(* Logix 5000 project; controller Savage_Saw vendor 1 type 14 code 152 rev 37.11; software revision 37.01 *)

TASK MainTask (continuous, watchdog 500 ms) : MainProgram, Inputs

MODULES
   Local : vendor 1 type 14 code 152 (PointIO 0, rev 37.11)
      Kane : vendor 590 type 43 code 5 (Ethernet 192.168.3.12, rev 1.1, StandardDataDriven RPI 20 ms, StandardDataDriven RPI 20 ms)
      RemoteHPU : 1734-AENTR (Ethernet 192.168.3.11, rev 7.13, Output RPI 20 ms)
         AnalogIn5_6 : 1734-IE2V (PointIO 1, rev 3.5, Input RPI 80 ms)
         InputDC0_8 : 1734-IB8 (PointIO 2, rev 3.22)
         InputDC9_15 : 1734-IB8 (PointIO 3, rev 3.1)
         OutputDC0_3 : vendor 1 type 7 code 134 (PointIO 5, rev 3.2)
         OutputDC4_7 : vendor 1 type 7 code 134 (PointIO 6, rev 3.2)
      Analog0_1 : 1734-IE2V (PointIO 2, rev 3.5, Input RPI 80 ms)
      Analog2_3 : 1734-IE2V (PointIO 3, rev 3.4, Input RPI 80 ms)
      Analog4_5 : 1734-IE2V (PointIO 4, rev 3.1, Input RPI 80 ms)
      Discrete_IO : Embedded (PointIO 1, rev 37.11, Output RPI 20 ms)
      SpindleControl : 1734-OE2V (PointIO 5, rev 3.1, Output RPI 80 ms)
       : 1734-OA4 (PointIO 6, rev 3.22, Output RPI 20 ms)
       : 1734-OA4 (PointIO 7, rev 3.1, Output RPI 20 ms)
       : 1734-OA4 (PointIO 8, rev 3.1, Output RPI 20 ms)
END_MODULES

TYPE AxisData :
STRUCT
   PositionActual : REAL;
   PositionCommand : REAL;
   VelocityCommand : REAL;
   InPosition : BOOL;
   AtVelocity : BOOL;
   OpenLoop : BOOL;
   FaultInput : BOOL;
   LimitPos : BOOL;
   LimitNeg : BOOL;
   Stopped : BOOL;
   InputEstimated : BOOL;
   OutputEnabled : BOOL;
   TargetGeneratorDone : BOOL;
   TargetGeneratorStateA : BOOL;
   TargetGeneratorStateB : BOOL;
   DirectOutput : BOOL;
   Enabled : BOOL;
   ExternalHalt : BOOL;
   Halted : BOOL;
   ForceControlled : BOOL;
   ForceLimitEnabled : BOOL;
   ForceLimited : BOOL;
   AtForce : BOOL;
   ForceInputEstimated : BOOL;
   ForceTargetGeneratorDone : BOOL;
   ForceTargetGeneratorStateA : BOOL;
   ForceTargetGeneratorStateB : BOOL;
   TargetGeneratorBusy : BOOL;
   ForceTargetGeneratorBusy : BOOL;
   FeedbackOK : BOOL;
   FeedbackOkSecondary : BOOL;
   StateMachineEnabled : BOOL;
   zs29 : BOOL;
   zs30 : BOOL;
   CommandAcknowledged : BOOL;
   CommandMove : BOOL;
   CommandJog : BOOL;
   Reverse : BOOL;
   z03 : BOOL;
   z04 : BOOL;
   z05 : BOOL;
   z06 : BOOL;
   z07 : BOOL;
   z08 : BOOL;
   z09 : BOOL;
   z10 : BOOL;
   z11 : BOOL;
   z12 : BOOL;
   z13 : BOOL;
   z14 : BOOL;
   z15 : BOOL;
   z16 : BOOL;
   z17 : BOOL;
   z18 : BOOL;
   z19 : BOOL;
   z20 : BOOL;
   z21 : BOOL;
   z22 : BOOL;
   z23 : BOOL;
   z24 : BOOL;
   z25 : BOOL;
   z26 : BOOL;
   z27 : BOOL;
   z28 : BOOL;
   z29 : BOOL;
   z30 : BOOL;
   z31 : BOOL;
END_STRUCT
END_TYPE

VAR_GLOBAL   (* controller tags *)
   Axis : AxisData[3];
   InBackGaugePot : ALIAS FOR Local:3:I.Ch1Data;
   inMS1HydraulicPump : ALIAS FOR Local:1:I.Data.1;
   inMS2HydraulicLoopPump : ALIAS FOR Local:1:I.Data.2;
   InMS3HydCoolingFan : ALIAS FOR Local:1:I.Data.3;
   inMS4CoolantPump : ALIAS FOR Local:1:I.Data.4;
   inMS5SwarfPump : ALIAS FOR Local:1:I.Data.5;
   inMS6SwarfConveyor : ALIAS FOR Local:1:I.Data.6;
   inRaiseLowerPot : ALIAS FOR Local:2:I.Ch1Data;
   inSpindleAside : ALIAS FOR Local:4:I.Ch0Data;
   inSpindleBside : ALIAS FOR Local:4:I.Ch1Data;
   inSpindleSpeed : ALIAS FOR Local:2:I.Ch0Data;
   inSR1SafetyRelay : ALIAS FOR Local:1:I.Data.0;
   inTraversePot : ALIAS FOR Local:3:I.Ch0Data;
   outLaserLine : ALIAS FOR Local:8:O.Data.0;
   outMS1HydraulicPump : ALIAS FOR Local:6:O.Data.0;
   outMS2HydraulicLoopPump : ALIAS FOR Local:6:O.Data.1;
   outMS3HydraulicCoolingFan : ALIAS FOR Local:6:O.Data.2;
   outMS4CoolantPump : ALIAS FOR Local:6:O.Data.3;
   outMS5SwarfPump : ALIAS FOR Local:7:O.Data.0;
   outMS6SwarfConveyor : ALIAS FOR Local:7:O.Data.1;
   outSpindleMotor : ALIAS FOR Local:5:O.Ch1Data;
   outSpindlePump : ALIAS FOR Local:5:O.Ch0Data;
   outStackLtAmber : ALIAS FOR Local:8:O.Data.2;
   outStackLtGreen : ALIAS FOR Local:8:O.Data.1;
   outStackLtRed : ALIAS FOR Local:8:O.Data.3;
   tbA1JogIn : BOOL;
   tbA1JogOut : BOOL;
   tbA2JogMinus : BOOL;
   tbA3JogMinus : BOOL;
   tbA3JogPlus : BOOL;
   tbAutoCut : BOOL;
   tbAutoGage : BOOL;
   tbAutoWet : BOOL;
   tbBladeChange : BOOL;
   tbBladeCompensation : BOOL;
   tbBladeMeasure : BOOL;
   tbCCW : BOOL;
   tbCoolant : BOOL;
   tbCW : BOOL;
   tbDryBump : BOOL;
   tbDryDist : BOOL;
   tbLaser : BOOL;
   tbMS1HydPump : BOOL;
   tbMS2LoopPump : BOOL;
   tbMS3HydCoolingFan : BOOL;
   tbMS4CoolantPump : BOOL;
   tbMS5SwarfPump : BOOL;
   tbMS6SwarfConveyor : BOOL;
   tbNorthRef : BOOL;
   tbOnOff : BOOL;
   tbPlateMeasure : BOOL;
   tbSouthRef : BOOL;
   tbWetBump : BOOL;
   tbWetDistance : BOOL;
   test : DINT;
   tmrTest : TIMER := (PRE := 1000);
   X_AutoCut : BOOL;
   X_AutoGauge : BOOL;
   X_BladeChange : BOOL;
   X_BladeMeasure : BOOL;
   X_Fault : BOOL;
   X_Homing : BOOL;
   X_Manual : BOOL;
   X_Off : BOOL;
END_VAR

PROGRAM Inputs   (* main routine Main *)

ROUTINE inAnalog   (* ladder *)
   0: ;
END_ROUTINE

ROUTINE Main   (* ladder *)
END_ROUTINE
END_PROGRAM

PROGRAM MainProgram   (* main routine Main *)
VAR
   iAxis : DINT;
END_VAR

ROUTINE Main   (* ladder *)
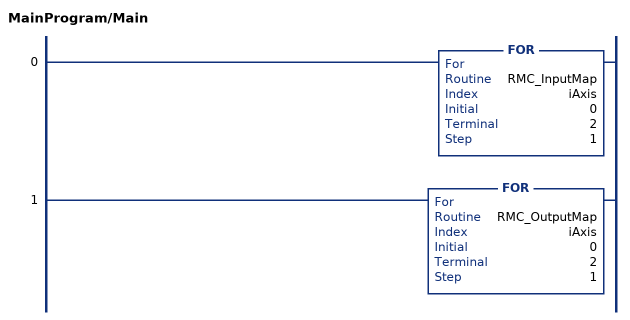
   0: FOR(RMC_InputMap,iAxis,0,2,1);
   1: FOR(RMC_OutputMap,iAxis,0,2,1);
END_ROUTINE

ROUTINE RMC_InputMap   (* ladder *)
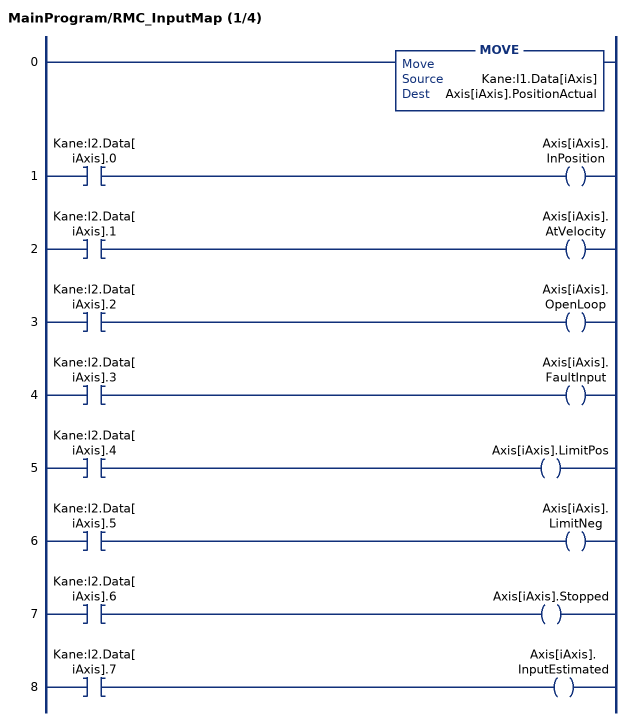
   0: MOVE(Kane:I1.Data[iAxis],Axis[iAxis].PositionActual);
   1: XIC(Kane:I2.Data[iAxis].0)OTE(Axis[iAxis].InPosition);
   2: XIC(Kane:I2.Data[iAxis].1)OTE(Axis[iAxis].AtVelocity);
   3: XIC(Kane:I2.Data[iAxis].2)OTE(Axis[iAxis].OpenLoop);
   4: XIC(Kane:I2.Data[iAxis].3)OTE(Axis[iAxis].FaultInput);
   5: XIC(Kane:I2.Data[iAxis].4)OTE(Axis[iAxis].LimitPos);
   6: XIC(Kane:I2.Data[iAxis].5)OTE(Axis[iAxis].LimitNeg);
   7: XIC(Kane:I2.Data[iAxis].6)OTE(Axis[iAxis].Stopped);
   8: XIC(Kane:I2.Data[iAxis].7)OTE(Axis[iAxis].InputEstimated);
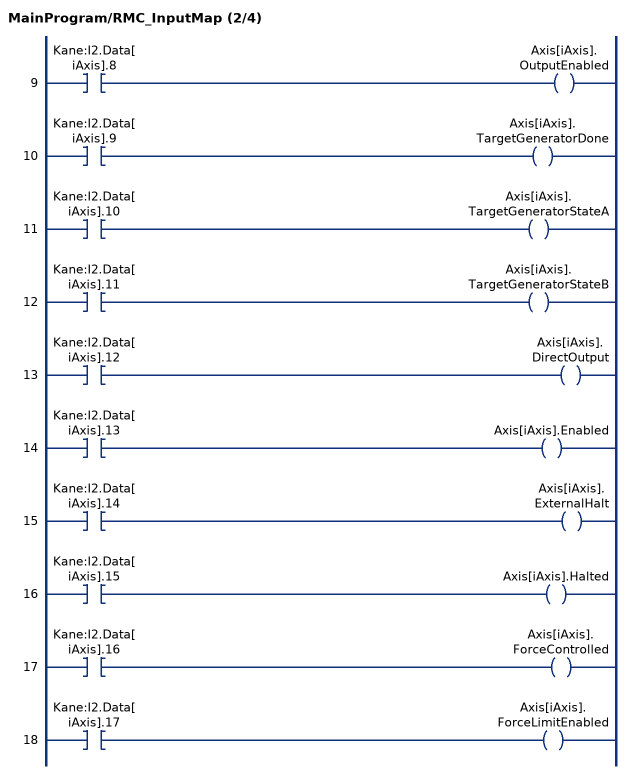
   9: XIC(Kane:I2.Data[iAxis].8)OTE(Axis[iAxis].OutputEnabled);
   10: XIC(Kane:I2.Data[iAxis].9)OTE(Axis[iAxis].TargetGeneratorDone);
   11: XIC(Kane:I2.Data[iAxis].10)OTE(Axis[iAxis].TargetGeneratorStateA);
   12: XIC(Kane:I2.Data[iAxis].11)OTE(Axis[iAxis].TargetGeneratorStateB);
   13: XIC(Kane:I2.Data[iAxis].12)OTE(Axis[iAxis].DirectOutput);
   14: XIC(Kane:I2.Data[iAxis].13)OTE(Axis[iAxis].Enabled);
   15: XIC(Kane:I2.Data[iAxis].14)OTE(Axis[iAxis].ExternalHalt);
   16: XIC(Kane:I2.Data[iAxis].15)OTE(Axis[iAxis].Halted);
   17: XIC(Kane:I2.Data[iAxis].16)OTE(Axis[iAxis].ForceControlled);
   18: XIC(Kane:I2.Data[iAxis].17)OTE(Axis[iAxis].ForceLimitEnabled);
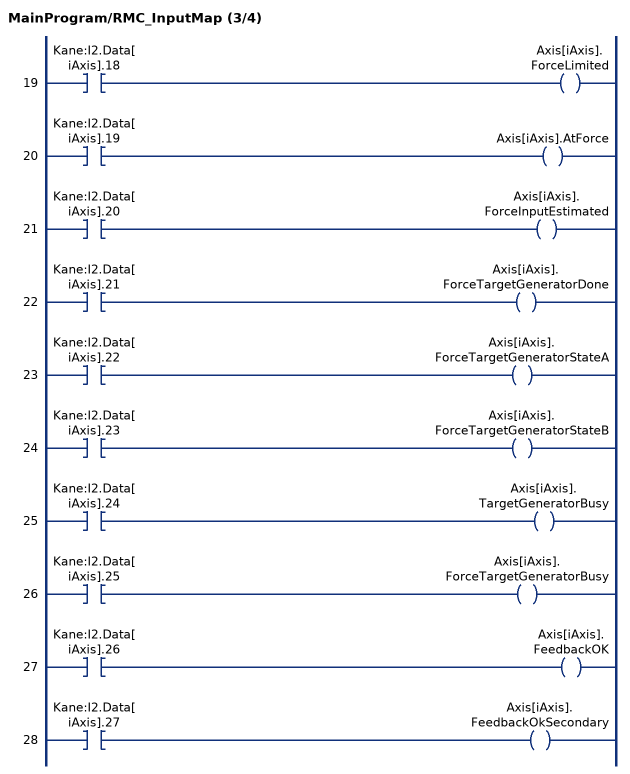
   19: XIC(Kane:I2.Data[iAxis].18)OTE(Axis[iAxis].ForceLimited);
   20: XIC(Kane:I2.Data[iAxis].19)OTE(Axis[iAxis].AtForce);
   21: XIC(Kane:I2.Data[iAxis].20)OTE(Axis[iAxis].ForceInputEstimated);
   22: XIC(Kane:I2.Data[iAxis].21)OTE(Axis[iAxis].ForceTargetGeneratorDone);
   23: XIC(Kane:I2.Data[iAxis].22)OTE(Axis[iAxis].ForceTargetGeneratorStateA);
   24: XIC(Kane:I2.Data[iAxis].23)OTE(Axis[iAxis].ForceTargetGeneratorStateB);
   25: XIC(Kane:I2.Data[iAxis].24)OTE(Axis[iAxis].TargetGeneratorBusy);
   26: XIC(Kane:I2.Data[iAxis].25)OTE(Axis[iAxis].ForceTargetGeneratorBusy);
   27: XIC(Kane:I2.Data[iAxis].26)OTE(Axis[iAxis].FeedbackOK);
   28: XIC(Kane:I2.Data[iAxis].27)OTE(Axis[iAxis].FeedbackOkSecondary);
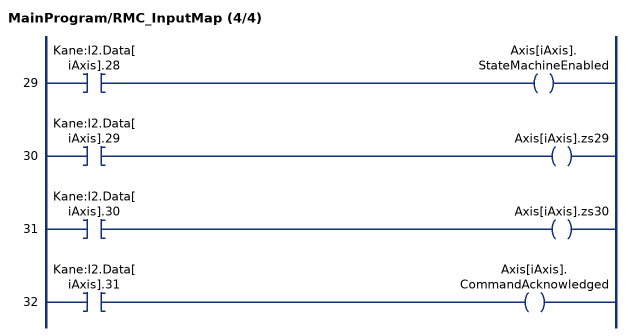
   29: XIC(Kane:I2.Data[iAxis].28)OTE(Axis[iAxis].StateMachineEnabled);
   30: XIC(Kane:I2.Data[iAxis].29)OTE(Axis[iAxis].zs29);
   31: XIC(Kane:I2.Data[iAxis].30)OTE(Axis[iAxis].zs30);
   32: XIC(Kane:I2.Data[iAxis].31)OTE(Axis[iAxis].CommandAcknowledged);
END_ROUTINE

ROUTINE RMC_OutputMap   (* ladder *)
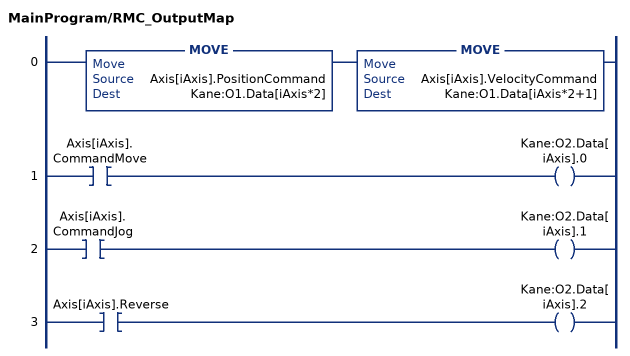
   0: MOVE(Axis[iAxis].PositionCommand,Kane:O1.Data[iAxis*2])MOVE(Axis[iAxis].VelocityCommand,Kane:O1.Data[iAxis*2+1]);
   1: XIC(Axis[iAxis].CommandMove)OTE(Kane:O2.Data[iAxis].0);
   2: XIC(Axis[iAxis].CommandJog)OTE(Kane:O2.Data[iAxis].1);
   3: XIC(Axis[iAxis].Reverse)OTE(Kane:O2.Data[iAxis].2);
END_ROUTINE
END_PROGRAM
